// TIA Portal project "109739660_Transport_V18" (V18)

(* hardware
DEVICE "S71500/ET200MP station_1"  S7-1500 station
   slot 0: "Rail_0"  Rack  6ES7 590-1***0-0AA0
   slot 1: "PLC_1"  CPU 1516-3 PN/DP  6ES7 516-3AN01-0AB0  V2.0
      slot 3: "CPU display_1"  6ES7591-1BA00-0AA0
DEVICE "HMI_1"  TP900 Comfort
   slot 0: "TP900 Comfort"  TP900 Comfort  6AV2 124-0JC01-0AX0  14.0.0.0
   slot 1: "HMI_RT_1"  TP900 Comfort  6AV2 124-0JC01-0AX0  14.0.0.0
   slot 5: "HMI_1.IE_CP_1"  PROFINET Interface  14.0.0.0
      slot 1: "PROFINET Interface_1"  PROFINET Interface
         slot 1: "Port_1"  Port
         slot 2: "Port_2"  Port
   slot 7: "HMI_1.MPI/DP_CP_1"  MPI/DP Interface  14.0.0.0
*)

// ===== PLC "PLC_1"  CPU 1516-3 PN/DP =====

VAR_GLOBAL   // PLC tag table "CommunicationWithCoSim"
   "sensorStartPos" AT %I0.0 : Bool;
   "sensorBeltStart" AT %I0.1 : Bool;
   "sensorBeltDest" AT %I0.2 : Bool;
   "sensorEndPos" AT %I0.3 : Bool;
   "setOnBeltActive" AT %Q0.0 : Bool;
   "moveBeltActive" AT %Q0.1 : Bool;
   "setOffBeltActive" AT %Q0.2 : Bool;
   "releaseActive" AT %Q0.3 : Bool;
   "acknowledgeActive" AT %Q0.4 : Bool;
   "restartActive" AT %Q0.5 : Bool;
END_VAR

VAR_GLOBAL   // PLC tag table "InternTags"
   "internAcknowledge" AT %M10.0 : Bool;
   "internRestart" AT %M10.1 : Bool;
END_VAR

DATA_BLOCK "Global"   // DB1
{ S7_Optimized_Access := 'TRUE' }
VERSION : 0.1
   VAR
      setOnBeltActive : Bool;
      moveBeltActive : Bool;
      setOffBeltActive : Bool;
      releaseActive : Bool;
      acknowledgeActive : Bool;
      restartActive : Bool;
      errorActive : Bool;
   END_VAR
BEGIN
END_DATA_BLOCK

DATA_BLOCK "InstTransport"   // DB2
{ S7_Optimized_Access := 'TRUE' }
VERSION : 0.1
// stored: InstanceOfName Transport
"Transport"
BEGIN
END_DATA_BLOCK

FUNCTION_BLOCK "Transport"   // FB1, GRAPH_PLUS
{ S7_Optimized_Access := 'TRUE' }
VERSION : 0.1
   VAR_INPUT
      OFF_SQ : Bool := false;   // Turn sequence off
      INIT_SQ : Bool := false;   // Set sequence to initial state
      ACK_EF : Bool := false;   // Acknowledge all errors and faults
      S_PREV : Bool := false;   // Output previous step in parameter S_NO
      S_NEXT : Bool := false;   // Indicate next step in parameter S_NO
      SW_AUTO : Bool := false;   // Automatic mode
      SW_TAP : Bool := false;   // Semiautomatic/switch with transition
      SW_TOP : Bool := false;   // Semiautomatic/ignore transition
      SW_MAN : Bool := false;   // Manual mode
      S_SEL : Int := 0;   // Select step to be output to S_NO
      S_ON : Bool := false;   // Activate step indicated in S_NO
      S_OFF : Bool := false;   // Deactivate step indicated S_NO
      T_PUSH : Bool := false;   // Enable transition to switch in semi automatic mode
   END_VAR
   VAR_OUTPUT
      S_NO : Int := 0;   // Step number
      S_MORE : Bool := false;   // More steps are available and can be shown in S_NO
      S_ACTIVE : Bool := false;   // Step indicated in S_NO is active
      ERR_FLT : Bool := false;   // Interlock or supervision group error
      AUTO_ON : Bool := false;   // Automatic mode is active
      TAP_ON : Bool := false;   // Semiautomatic mode/step with transition enabled
      TOP_ON : Bool := false;   // Semiautomatic mode/ignore transition enabled
      MAN_ON : Bool := false;   // Manual mode is active
   END_VAR
   VAR
      instMoveBelt : "MoveBelt";
      instSetOffBelt : "SetOffBelt";
      instSetOnBelt : "SetOnBelt";
      instRelease : "Release";
   END_VAR
   VAR RETAIN
      HMI_INFO : Array[0..8] of UInt;
      IF_PAR : G7_IfParPlus_V3;
      RT_DATA : G7_RTDataPlus_V3;   // Internal data area
      "Package reaches start position" : G7_TransitionPlus_V3;   // Transition structure
      "Package reaches belt start position" : G7_TransitionPlus_V3;   // Transition structure
      "Package reaches belt destination position" : G7_TransitionPlus_V3;   // Transition structure
      "Package reaches end position" : G7_TransitionPlus_V3;   // Transition structure
      "Package left end position" : G7_TransitionPlus_V3;   // Transition structure
      "Check package at start position" : G7_StepPlus_V3;   // Step structure
      "Set package on belt" : G7_StepPlus_V3;   // Step structure
      "Move Belt" : G7_StepPlus_V3;   // Step structure
      "Set package off belt" : G7_StepPlus_V3;   // Step structure
      "Release package" : G7_StepPlus_V3;   // Step structure
      SINI : Array[0..1] of USInt;
      LSTT : Array[0..4] of USInt;
      ATAJ : Array[0..4] of USInt;
      ATAB : Array[0..4] of USInt;
      PSTT : Array[0..4] of USInt;
      NSTT : Array[0..4] of USInt;
      ASSJ : Array[0..4] of USInt;
      ASSB : Array[0..4] of USInt;
      PTTS : Array[0..4] of USInt;
      NTTS : Array[0..4] of USInt;
      SW_SQTS : Array[0..4] of USInt;
      SWITCH : Array[0..0] of USInt;
      TVX : Array[0..1] of USInt;
      TTX : Array[0..1] of USInt;
      TSX : Array[0..1] of USInt;
      S00X : Array[0..1] of USInt;
      SOFFX : Array[0..1] of USInt;
      SONX : Array[0..1] of USInt;
      SAX : Array[0..1] of USInt;
      SERRX : Array[0..5] of USInt;
      SMX : Array[0..5] of USInt;
      S0X : Array[0..5] of USInt;
      S1X : Array[0..5] of USInt;
      IL_ALARM_INST : Diag_Alarm;
      SUP_ALARM_INST : Diag_Alarm;
      STEP_TIME_ALARM_INST : Diag_Alarm;
      IEC_TIMER_INST : IEC_TIMER;
   END_VAR
   VAR CONSTANT
      TIME_CHECK : Time := T#5000ms;   // Supervision time for step 3 (Move belt)
   END_VAR
   // SINI[0] := 2;
   // LSTT[0] := 255;
   // LSTT[1] := 255;
   // LSTT[2] := 255;
   // LSTT[3] := 255;
   // ATAJ[1] := 1;
   // ATAJ[2] := 2;
   // ATAJ[3] := 3;
   // ATAJ[4] := 4;
   // ATAB[1] := 1;
   // ATAB[2] := 2;
   // ATAB[3] := 3;
   // ATAB[4] := 4;
   // PSTT[1] := 1;
   // PSTT[2] := 2;
   // PSTT[3] := 3;
   // PSTT[4] := 4;
   // NSTT[0] := 1;
   // NSTT[1] := 2;
   // NSTT[2] := 3;
   // NSTT[3] := 4;
   // ASSJ[1] := 1;
   // ASSJ[2] := 2;
   // ASSJ[3] := 3;
   // ASSJ[4] := 4;
   // ASSB[1] := 1;
   // ASSB[2] := 2;
   // ASSB[3] := 3;
   // ASSB[4] := 4;
   // PTTS[0] := 255;
   // PTTS[2] := 1;
   // PTTS[3] := 2;
   // PTTS[4] := 3;
   // NTTS[1] := 1;
   // NTTS[2] := 2;
   // NTTS[3] := 3;
   // NTTS[4] := 4;
   // TVX[0] := 16#1;
   // TTX[0] := 16#1;
   // TSX[0] := 16#1;
   // S00X[0] := 16#1;
   // SOFFX[0] := 16#1;
   // SONX[0] := 16#1;
   // SAX[0] := 16#1;
   // SERRX[0] := 16#1;
   // SMX[0] := 16#1;
   // S0X[0] := 16#1;
   // S1X[0] := 16#1;
BEGIN
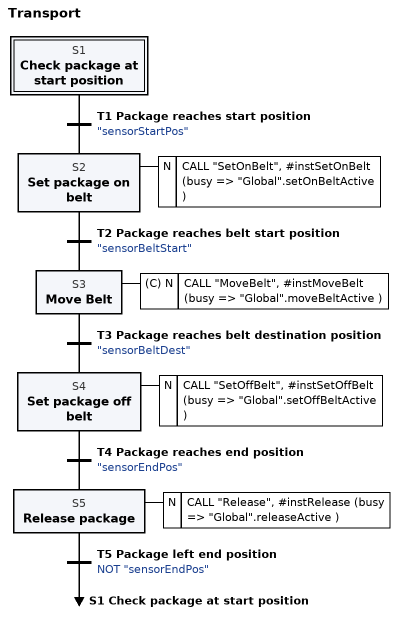
   // sequencer 1
   INITIAL_STEP "Check package at start position":   // S1, max time T#10S, warning time T#7S
      interlock C := (none);   // -
      supervision V := (none);   // -
      // No Action (Idle). Waiting for the package. / -
   END_STEP
   TRANSITION "Package reaches start position" FROM "Check package at start position" TO "Set package on belt"   // T1: -
      := "sensorStartPos";
   END_TRANSITION
   STEP "Set package on belt":   // S2, max time T#10S, warning time T#7S
      interlock C := (none);   // -
      supervision V := (none);   // -
      // Call the function block "SetOnBelt" / -
              N    CALL "SetOnBelt", #instSetOnBelt
                   (busy => "Global".setOnBeltActive
                   )
   END_STEP
   TRANSITION "Package reaches belt start position" FROM "Set package on belt" TO "Move Belt"   // T2: -
      := "sensorBeltStart";
   END_TRANSITION
   STEP "Move Belt":   // S3, max time T#10S, warning time T#7S
      interlock C := NOT #"Move Belt".VA;   // Check Error
      supervision V := #"Move Belt".T > #TIME_CHECK;   // Check package reach belt destination position on time
      // Call function block "MoveBelt". / -
      (C)     N    CALL "MoveBelt", #instMoveBelt
                   (busy => "Global".moveBeltActive
                   )
   END_STEP
   TRANSITION "Package reaches belt destination position" FROM "Move Belt" TO "Set package off belt"   // T3
      := "sensorBeltDest";
   END_TRANSITION
   STEP "Set package off belt":   // S4, max time T#10S, warning time T#7S
      interlock C := (none);   // -
      supervision V := (none);   // -
      // Call function block "SetOff Belt".
              N    CALL "SetOffBelt", #instSetOffBelt
                   (busy => "Global".setOffBeltActive
                   )
   END_STEP
   TRANSITION "Package reaches end position" FROM "Set package off belt" TO "Release package"   // T4
      := "sensorEndPos";
   END_TRANSITION
   STEP "Release package":   // S5, max time T#10S, warning time T#7S
      interlock C := (none);   // -
      supervision V := (none);   // -
      // Call function block "Release"
              N    CALL "Release", #instRelease
                   (busy => "Global".releaseActive
                   )
   END_STEP
   TRANSITION "Package left end position" FROM "Release package" TO "Check package at start position"   // T5, jump
      := NOT "sensorEndPos";
   END_TRANSITION
END_FUNCTION_BLOCK

FUNCTION "Initialize" : Void   // FC1, SCL
{ S7_Optimized_Access := 'TRUE' }
VERSION : 0.1
BEGIN
   // Inititialize global variables

   "Global".setOnBeltActive := 0;
   "Global".moveBeltActive := 0;
   "Global".setOffBeltActive := 0;
   "Global".releaseActive := 0;
END_FUNCTION

FUNCTION "ReadInputs" : Void   // FC2, SCL
{ S7_Optimized_Access := 'TRUE' }
VERSION : 0.1
BEGIN
   // Read inputs from HMI

   "Global".acknowledgeActive := "internAcknowledge";
   "Global".restartActive := "internRestart";
END_FUNCTION

FUNCTION "WriteOtputs" : Void   // FC3, SCL
{ S7_Optimized_Access := 'TRUE' }
VERSION : 0.1
BEGIN
   // Write outputs for Co-Simulation
   "setOnBeltActive" := "Global".setOnBeltActive;
   "moveBeltActive" := "Global".moveBeltActive;
   "setOffBeltActive" := "Global".setOffBeltActive;
   "releaseActive" := "Global".releaseActive;

   "acknowledgeActive" := "Global".acknowledgeActive;
   "restartActive" := "Global".restartActive;
END_FUNCTION

ORGANIZATION_BLOCK "Main"   // OB1, LAD, ProgramCycle
TITLE = "Main Program Sweep (Cycle)"
{ S7_Optimized_Access := 'TRUE' }
VERSION : 0.1
   VAR_INPUT
      Initial_Call : Bool;   // Initial call of this OB
      Remanence : Bool;   // =True, if remanent data are available
   END_VAR
BEGIN

REGION Network 1: Initialize global variables
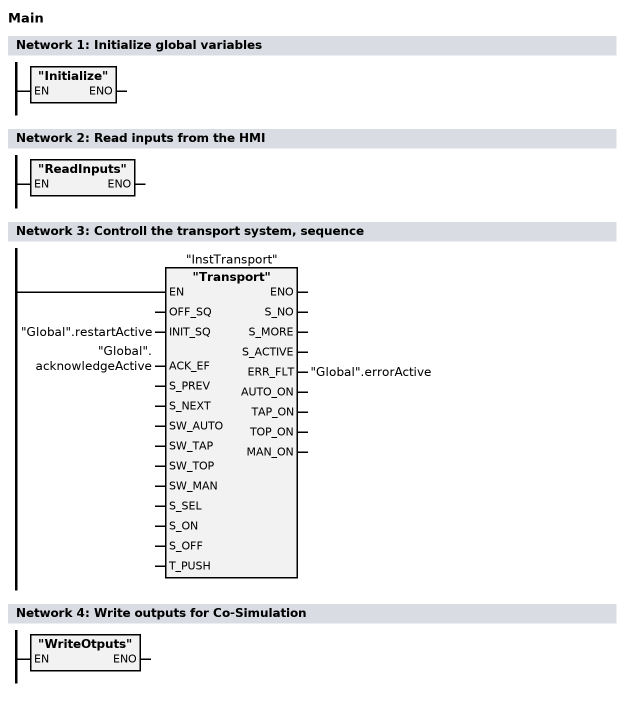
   RUNG wire#powerrail
      "Initialize"()
   END_RUNG
   // the same network as SCL:
   "Initialize"();
END_REGION

REGION Network 2: Read inputs from the HMI
   RUNG wire#powerrail
      "ReadInputs"()
   END_RUNG
   // the same network as SCL:
   "ReadInputs"();
END_REGION

REGION Network 3: Controll the transport system, sequence
   RUNG wire#powerrail
      "InstTransport"(OFF_SQ :=, INIT_SQ := "Global".restartActive, ACK_EF := "Global".acknowledgeActive, S_PREV :=, S_NEXT :=, SW_AUTO :=, SW_TAP :=, SW_TOP :=, SW_MAN :=, S_SEL :=, S_ON :=, S_OFF :=, T_PUSH :=, S_NO =>, S_MORE =>, S_ACTIVE =>, ERR_FLT => "Global".errorActive, AUTO_ON =>, TAP_ON =>, TOP_ON =>, MAN_ON =>)
   END_RUNG
   // the same network as SCL:
   "InstTransport"(INIT_SQ := "Global".restartActive,   // "Transport"
                   ACK_EF := "Global".acknowledgeActive,
                   ERR_FLT => "Global".errorActive);
END_REGION

REGION Network 4: Write outputs for Co-Simulation
   RUNG wire#powerrail
      "WriteOtputs"()
   END_RUNG
   // the same network as SCL:
   "WriteOtputs"();
END_REGION
END_ORGANIZATION_BLOCK

// folder: TransportFunctions

FUNCTION_BLOCK "MoveBelt"   // FB2, SCL
{ S7_Optimized_Access := 'TRUE' }
VERSION : 0.1
   VAR_OUTPUT
      busy : Bool;
   END_VAR
BEGIN
   // Dummy function
   // When function block is called, output "busy" is set.

   #busy := 1;
END_FUNCTION_BLOCK

FUNCTION_BLOCK "Release"   // FB3, SCL
{ S7_Optimized_Access := 'TRUE' }
VERSION : 0.1
   VAR_OUTPUT
      busy : Bool;
   END_VAR
BEGIN
   // Dummy function
   // When function block is called, output "busy" is set.

   #busy := 1;
END_FUNCTION_BLOCK

FUNCTION_BLOCK "SetOffBelt"   // FB4, SCL
{ S7_Optimized_Access := 'TRUE' }
VERSION : 0.1
   VAR_OUTPUT
      busy : Bool;
   END_VAR
BEGIN
   // Dummy function
   // When function block is called, output "busy" is set.

   #busy := 1;
END_FUNCTION_BLOCK

FUNCTION_BLOCK "SetOnBelt"   // FB5, SCL
{ S7_Optimized_Access := 'TRUE' }
VERSION : 0.1
   VAR_OUTPUT
      busy : Bool;
   END_VAR
BEGIN
   // Dummy function
   // When function block is called, output "busy" is set.

   #busy := 1;
END_FUNCTION_BLOCK

// ===== library types =====

// folder: 7 Signal generators

FUNCTION_BLOCK "LGF_Frequency"   // FB10024, SCL
{ S7_Optimized_Access := 'TRUE' }
   VAR_INPUT
      frequency : Real;   // Input in Hz
   END_VAR
   VAR_OUTPUT
      clock : Bool;
      countdown : Time;
   END_VAR
   VAR
      instTofTimeOn : TOF_TIME;
      instTofTimeOff : TOF_TIME;
      statFrequencyMem : Real;
      statTimeBase : Time;
   END_VAR
   VAR CONSTANT
      NULL : Real := 0.0;
   END_VAR
BEGIN
   //=============================================================================
   // SIEMENS AG
   // (c)Copyright 2015
   //-----------------------------------------------------------------------------
   // Library:       LGF(Library General Functions)
   // Tested with:   CPU1212C DC/DC/DC FW:V4.1
   // Engineering:   TIA Portal V13 SP1 Upd 4
   // Restrictions:  -
   // Requirements:  PLC (S7-1200, S7-1500)
   // Functionality: Generates frequency signal
   //-----------------------------------------------------------------------------
   // Change log table:
   // Version  Date        Expert in charge                Changes applied
   // 01.00.00 19.08.2015  Siemens Industry Online Support First released version 
   //=============================================================================

   IF (#frequency <= #NULL)  // If input is <= 0.0 >> block is off // Wenn Eingang kleiner als 0.0 >> Baustein arbeitet nicht
   THEN
     #clock := FALSE;
     #countdown := t#0s;
   ELSE
     IF #statFrequencyMem <> #frequency THEN // assign frequency one time   // Frequenz zuweisen
       #statTimeBase := t#1000s / TRUNC(#frequency * 2000); // calculate time  //Zeit berechnen
       #statFrequencyMem := #frequency;
     END_IF;

     // TOF_off expired >> Start again // TOF_off abgelaufen starte von vorn
     #instTofTimeOn(IN := NOT #instTofTimeOff.Q,
                    PT := #statTimeBase);
     #countdown := #statTimeBase - #instTofTimeOn.ET;

     #instTofTimeOff(IN := #instTofTimeOn.Q,
                     PT := #statTimeBase);

     IF #countdown = t#0s THEN
       #countdown := #statTimeBase - #instTofTimeOff.ET;
     END_IF;

     #clock := #instTofTimeOn.Q; //assign ouptut // Frequenzausgang setzen   
   END_IF;
END_FUNCTION_BLOCK

(* ===== HMI "HMI_RT_1" =====
system functions are stored by id; their names below are inferred from use
connection "HMI_Connection_1": ETHERNET, S7_1500_OMS

HMI tags "DefaultTagTable"
   "globalErrorActive" : Bool = PLC Global.errorActive AT %DB1.DBX0.0, 100 ms
   "internAcknowledge" : Bool = PLC internAcknowledge AT %M10.0, 100 ms
   "internRestart" : Bool = PLC internRestart AT %M10.1, 100 ms
   "moveBeltActive" : Bool = PLC moveBeltActive AT %Q0.1, 100 ms
   "releaseActive" : Bool = PLC releaseActive AT %Q0.3, 100 ms
   "sensorBeltDest" : Bool = PLC sensorBeltDest AT %I0.2, 100 ms
   "sensorBeltStart" : Bool = PLC sensorBeltStart AT %I0.1, 100 ms
   "sensorEndPos" : Bool = PLC sensorEndPos AT %I0.3, 100 ms
   "sensorStartPos" : Bool = PLC sensorStartPos AT %I0.0, 100 ms
   "setOffBeltActive" : Bool = PLC setOffBeltActive AT %Q0.2, 100 ms
   "setOnBeltActive" : Bool = PLC setOnBeltActive AT %Q0.0, 100 ms

screen "RootScreen" 800x480, template "Template_1"
   GraphicView "Graphic view_1" at 23,184 size 124x17; Picture "conveyor_klein"
   GraphicView "Graphic view_3" at 228,184 size 320x17; Picture "conveyor_white"
      Visibility <- "moveBeltActive"
   GraphicView "Graphic view_5" at 633,184 size 124x17; Picture "conveyor_klein_white"
      Visibility <- "releaseActive"
   GraphicView "Graphic view_12" at 157,68 size 126x126; Picture "Robot_G_SY02_XX_01127_Green"
      Visibility <- "setOnBeltActive"
   GraphicView "Graphic view_14" at 558,68 size 126x126; Picture "Robot_G_SY02_XX_01127_Green"
      Visibility <- "setOffBeltActive"
   GraphicView "Graphic view_2" at 228,184 size 320x17; Picture "conveyor_black"
   GraphicView "Graphic view_4" at 633,184 size 124x17; Picture "conveyor_klein_black"
   GraphicView "Graphic view_6" at 22,201 size 24x69; Picture "Graphic_1"
   GraphicView "Graphic view_7" at 121,201 size 24x69; Picture "Graphic_1"
   GraphicView "Graphic view_8" at 227,201 size 24x69; Picture "Graphic_1"
   GraphicView "Graphic view_9" at 520,201 size 24x69; Picture "Graphic_1"
   GraphicView "Graphic view_10" at 632,201 size 24x69; Picture "Graphic_1"
   GraphicView "Graphic view_11" at 732,201 size 24x69; Picture "Graphic_1"
   GraphicView "Graphic view_13" at 157,68 size 126x126; Picture "Robot_G_SY02_XX_01127"
   GraphicView "Graphic view_15" at 558,68 size 126x126; Picture "Robot_G_SY02_XX_01127"
   GraphicView "Graphic view_16" at 70,134 size 69x45; Picture "cargobox_blue"
      Visibility <- "sensorStartPos"
   GraphicView "Graphic view_17" at 643,134 size 69x45; Picture "cargobox_blue"
      Visibility <- "sensorEndPos"
   GraphicView "Graphic view_18" at 467,134 size 69x45; Picture "cargobox_blue"
      Visibility <- "sensorBeltDest"
   GraphicView "Graphic view_19" at 239,134 size 69x45; Picture "cargobox_blue"
      Visibility <- "sensorBeltStart"
   GraphicView "Graphic view_20" at 347,251 size 69x45; Picture "cargobox_red"
      Visibility <- "globalErrorActive"
   TextField "Text field_1" at 302,222 size 159x20; Text 'Error: Package down'
      Visibility <- "globalErrorActive"
   Button "Button_1" at 474,324 size 136x60; TextOff 'Acknowledge'
      on Press: SetBit("internAcknowledge")
      on Release: ResetBit("internAcknowledge")
   Button "Button_2" at 631,324 size 136x60; TextOff 'Restart'
      on Press: SetBit("internRestart")
      on Release: ResetBit("internRestart")
   GraphicView "Graphic view_21" at 353,134 size 69x45; Picture "cargobox_blue"
      Visibility <- "moveBeltActive"

Template "Template_1" 800x480
   Button "Exit" at 720,420 size 78x58; TextOff 'Exit'; PictureOff "ExitRuntime_TP900_Comfort_TR"; PictureOn "ExitRuntime_TP900_Comfort_TR"
      on Release: StopRuntime(0)
   Button "Template_Button" at 640,420 size 78x58; TextOff 'Text'
   Button "Template_Button_1" at 560,420 size 78x58; TextOff 'Text'
   Button "Template_Button_2" at 480,420 size 78x58; TextOff 'Text'
   Button "Template_Button_3" at 400,420 size 78x58; TextOff 'Text'
   Button "Template_Button_4" at 320,420 size 78x58; TextOff 'Text'
   Button "Template_Button_5" at 240,420 size 78x58; TextOff 'Text'
   Button "Template_Button_6" at 160,420 size 78x58; TextOff 'Text'
   Button "Alarms" at 80,420 size 78x58; TextOff 'Alarms'; PictureOff "AlarmDisplay_TP900_Comfort_TR"; PictureOn "AlarmDisplay_TP900_Comfort_TR"
      on Release: function_ef3f5d25("Alarm window_Unacknowledged", -1)
   Button "Start screen" at 1,420 size 78x58; TextOff 'Start screen'; PictureOff "NavigateHome_TP900_Comfort_TR"; PictureOn "NavigateHome_TP900_Comfort_TR"
      on Release: ActivateScreen("RootScreen", 0)
*)